// TwinCAT 3 PLC project TEXXX_XXX
// ProgramVersion: 3.1.4024.0
// libraries:
//   Tc2_Standard, * (Beckhoff Automation GmbH)
//   Tc2_System, * (Beckhoff Automation GmbH)
//   Tc2_Utilities, * (Beckhoff Automation GmbH)
//   Tc3_Module, * (Beckhoff Automation GmbH)
// project tree:
//   DUTs/HMI/ ST_StatusBanner.TcDUT (not stored), ST_Timers.TcDUT (not stored)
//   DUTs/IO/CARDS/ ST_Terminal_Info.TcDUT (not stored), ST_EL1809.TcDUT (not stored), ST_EL2809.TcDUT (not stored)
//   DUTs/MASTER/ E_MachineState.TcDUT (not stored), E_ProcessCycle.TcDUT (not stored), ST_ButtonsLamps.TcDUT (not stored), ST_HMI_IO.TcDUT (not stored), ST_MachineStatus.TcDUT (not stored), ST_MasterCTRL.TcDUT (not stored), ST_StationCMD.TcDUT (not stored), ST_StationStatus.TcDUT (not stored), ST_Puls.TcDUT (not stored), ST_StatisticsHMI.TcDUT (not stored)
//   DUTs/MASTER/log_CSV/ ST_CSVProcess.TcDUT, ST_UserLog.TcDUT (not stored), ST_CycleData.TcDUT (not stored)
//   DUTs/PDFMaker/ ST_EventsPDF.TcDUT, ST_EventsPdfConstants.TcDUT, ST_JavasCriptPDF.TcDUT, ST_PDFMaker.TcDUT
//   DUTs/STATIONS/STATION_1/ E_Station1_State.TcDUT (not stored), ST_CycleDataStation1.TcDUT (not stored), ST_Station_1.TcDUT (not stored)
//   DUTs/STATIONS/STATION_2/ E_Station2_State.TcDUT (not stored), ST_CycleDataStation2.TcDUT (not stored), ST_Station_2.TcDUT (not stored)
//   DUTs/STATIONS/STATION_3/ E_Station3_State.TcDUT (not stored), ST_CycleDataStation3.TcDUT (not stored), ST_Station_3.TcDUT (not stored)
//   DUTs/USER_ALARMS_EVENTS/EVENTS/ ST_ActiveEvents.TcDUT (not stored), ST_EventsAssigment.TcDUT (not stored), ST_EventsAssigmentGeneral.TcDUT (not stored), ST_EventsHistory.TcDUT, ST_EVENT.TcDUT (not stored), ST_StationEvents.TcDUT (not stored)
//   DUTs/USER_ALARMS_EVENTS/ ST_UserLogHMI.TcDUT (not stored)
//   GVLs/ GVL_Constants.TcGVL, GVL_HMI.TcGVL, GVL_IO.TcGVL (not stored), GVL_Master.TcGVL, GVL_Persistent.TcGVL, GVL_Stations.TcGVL (not stored)
//   / PlcTask.TcTTO (not stored)
//   POUs/A_MASTER/ A_1_PRG_Main_Master.TcPOU, A_2_PRG_MachineCtrl.TcPOU (not stored), A_3_PRG_FaultHandling.TcPOU (not stored), A_4_PRG_MasterSystemTime.TcPOU (not stored)
//   POUs/B_STATIONS/B_1_LEAK_TEST/ B_1_1_PRG_Master_Station_1.TcPOU (not stored)
//   POUs/B_STATIONS/B_2_HEIGHT_TEST/ B_2_1_PRG_Master_Station_2.TcPOU
//   POUs/B_STATIONS/B_3_STATION_3/ B_3_1_PRG_Master_Station_3.TcPOU (not stored)
//   POUs/C_HMI/ C_1_PRG_MainHMI.TcPOU (not stored)
//   POUs/ MAIN.TcPOU (not stored)
//   POUs/Utilities/ FB_EventsManager.TcPOU, FB_PDFMaker.TcPOU, FB_UserLog.TcPOU (not stored), FB_Pulse.TcPOU (not stored), FB_TerminalInfo.TcPOU (not stored), FB_TimeControl.TcPOU (not stored), FB_WriteDataToCSV.TcPOU, PRG_Puls.TcPOU (not stored)
// real-time tasks:
//   TASK PlcTask: cycle T#10ms, priority 20, ADS port 350

// ---- DUTs/MASTER/log_CSV/ST_CSVProcess.TcDUT
TYPE ST_CSVProcess :
STRUCT
	
	//INPUTS
	bWriteData			: BOOL;
	bWriteCSV			: BOOL;
	sFileNamePath		: STRING(255);
	sDate				: STRING(255);
	aDataHistoryArrayLength : DINT;
	nMAX_CSV_ROWS		: UDINT;
	nMAX_CSV_COLUMNS	: UDINT;

	//OUTPUTS
	bError				: BOOL;
	bBusy				: BOOL;
	
	
	
	
END_STRUCT
END_TYPE

// ---- DUTs/PDFMaker/ST_EventsPDF.TcDUT
TYPE ST_EventsPDF :
STRUCT
	
	     sEvents				: STRING;
         sType					: STRING;
         sDate					: STRING;
         sTime					: STRING;

	
END_STRUCT
END_TYPE

// ---- DUTs/PDFMaker/ST_EventsPdfConstants.TcDUT
TYPE ST_EventsPdfConstants :
STRUCT
	
	sMachineName			: STRING(255);
	sUser					: STRING(255);
	sGroup					: STRING(255);
	sFileName				: STRING(255);
	
END_STRUCT
END_TYPE

// ---- DUTs/PDFMaker/ST_JavasCriptPDF.TcDUT
TYPE ST_JavasCriptPDF :
STRUCT
	
	stEventsPDF				: ARRAY [0..2000] OF ST_EventsPDF;
	stEventsPdfConstants	: ST_EventsPdfConstants;
	bMakePDF				: BOOL;
	
	
END_STRUCT
END_TYPE

// ---- DUTs/PDFMaker/ST_PDFMaker.TcDUT
TYPE ST_PDFMaker :
STRUCT
	
	//INPUTS
	bWriteData			: BOOL;
	sDate				: STRING(255);
	aDataHistoryArrayLength : DINT;
	nDataHistoryIndex	: DINT;
	

	//OUTPUTS
	
	sFileName			: STRING(255);
	bDataWrited			: BOOL;
	

END_STRUCT
END_TYPE

// ---- DUTs/USER_ALARMS_EVENTS/EVENTS/ST_EventsHistory.TcDUT
TYPE ST_EventsHistory :
STRUCT
	
	sEventTex									: STRING(255);
	sType										: STRING(255);
	sDate										: STRING(255);
	sTime										: STRING(255);
	nEventsAmount								: DINT;
	abType										: DINT;					//1:Alarm
																		//2:Alert
																		//3:Message
	
END_STRUCT
END_TYPE

// ---- GVLs/GVL_Constants.TcGVL
VAR_GLOBAL CONSTANT
////////////////////////////////////////:	///////////////////////////////////////////////////
/////////////////////////////////////////////////////////////////////////////////////HMI/////////////////////////////////////////////////////////////////////////////////////
	
    sWHITE                              :   STRING(40)  := '{"color":"rgba(255,255,255,255)"}';
    sBLACK                              :   STRING(40)  := '{"color":"rgba(0,0,0,1)"}';
    sYELLOW                             :   STRING(40)  := '{"color":"rgba(255,255,0,1)"}';
    sGREEN                             	:   STRING(40)  := '{"color":"rgba(70,166,63,1)"}';
	sLGREEN                             :   STRING(40)  := '{"color":"rgba(58,211,20,1)"}';
    sORANGE                             :   STRING(40)  := '{"color":"rgba(255,153,51,1)"}';
    sNYPROORANGE                        :   STRING(40)  := '{"color":"rgba(255,140,0,1)"}';
    sRED                                :   STRING(40)  := '{"color":"rgba(255,0,0,1)"}';
	sLRED                               :   STRING(40)  := '{"color":"rgba(233,53,44,1)"}';
    sBLUE                               :   STRING(40)  := '{"color":"rgba(0,0,255,1)"}';
	sLBLUE                              :   STRING(40)  := '{"color":"rgba(0,162,232,1)"}';
    sGREY                               :   STRING(40)  := '{"color":"rgba(164,158,158,1)"}';
    sScreenGREY                         :   STRING(40)  := '{"color":"rgba(225,225,225,1)"}';
    sDARKGREY                           :   STRING(40)  := '{"color":"rgba(50,50,50,1)"}';
    sPURPLE                             :   STRING(40)  := '{"color":"rgba(128,0,128,1)"}';
    sVIOLET                             :   STRING(40)  := '{"color":"rgba(204,153,255,1)"}';
    sTRANSP                             :   STRING(40)  := '{"color":"rgba(255,255,255,0)"}';
    sGREENPass                          :   STRING(40)  := '{"color":"rgba(0,153,51,1)"}';
    sREDFail                            :   STRING(40)  := '{"color":"rgba(244,68,68,255)"}';
    sBLUEInProgress                     :   STRING(40)  := '{"color":"rgba(54,100,221,1)"}';
	sGREENISHTEAColor					:	STRING(40)  := '{"color":"rgba(60,192,134,255)"}'	;		

	nBLACK								: 	DWORD 	:= 	16#FF000000;	 // format: TTRRGGBB where T -> 00 = full transparency and FF = full opaque
	nWHITE								: 	DWORD 	:= 	16#FFFFFFFF;
	nYELLOW								: 	DWORD 	:= 	16#FFFFFF00; 
	nGREEN								: 	DWORD 	:= 	16#FF008A00;
	nLIGHTGREEN                         :   DWORD   :=  16#FF98FB89;
	nORANGE								: 	DWORD 	:= 	16#FFFFA500;
	nNYPROORANGE						:	DWORD	:=	16#FFF05322;
	nRED								: 	DWORD 	:= 	16#FFFF0000;
	nBLUE								: 	DWORD 	:= 	16#FF0000FF;
	nLIGHTBLUE                          :   DWORD   :=  16#FF08ADF4;
	nGREY								: 	DWORD 	:= 	16#FFA9A9A9;	
	nDARKGREY							:	DWORD	:=	16#FF808080;
	nPURPLE								:	DWORD	:=	16#FF800080;
	nVIOLET								:	DWORD	:=	16#FFEE82EE;
	nTRANSP								:	DWORD	:=	16#00FFFFFF;	// full transparent WHITE
	
/////////////////////////////////////////////////////////////////////////////////////CSV/////////////////////////////////////////////////////////////////////////////////////
	

	
	
	
END_VAR

// ---- GVLs/GVL_HMI.TcGVL
VAR_GLOBAL
////////////////////////////////////////:	///////////////////////////////////////////////////
/////////////////////////////////////////////////////////////////////////////////////GENERIC/////////////////////////////////////////////////////////////////////////////////////

	stHMI_IO							: ST_HMI_IO;
	bQuitHMI							: BOOL;
	bShutDown							: BOOL;
	stStatusBanner						: ST_StatusBanner;
	rOpenPopUp							: R_TRIG;
	nPopUp								: DINT;
	
	

/////////////////////////////////////////////////////////////////////////////////////SYSTEM INFO/////////////////////////////////////////////////////////////////////////////////////

	sSoftwareVersion					: STRING := ' 1.0 ';
	sSoftwareDate						: STRING := ' 10.December.2024 ';
	sTC3Version							: STRING := ' v3.1.4024.53, Runtime v3.1.4024.40 ';
	sHMIVersion							: STRING := ' TcXaeShell Version 15.0.28010.2050 D15.8 ';
	sSystemName							: STRING := ' Print & Applay Labeller ' ;
	sProjectID							: STRING := ' TE 1099 PAL' ;
	sAplication                     	: STRING := ' Print & Applay Labeller ';
	sHMIServer                			: STRING := ' ---- ';
	
	NetAmsId        	       			: T_AmsNetId := ''; // AMS-ID for com port setup 
	
/////////////////////////////////////////////////////////////////////////////////////USER LOG/////////////////////////////////////////////////////////////////////////////////////

	sUserGroupIn						: STRING;
	sUserGroupOut						: STRING;
	sUserName							: STRING;
	bUserLoggedIn						: BOOL;			
	bLogOut								: BOOL;	
	rUserLoggedIn						: R_TRIG;

/////////////////////////////////////////////////////////////////////////////////////MANUAL/////////////////////////////////////////////////////////////////////////////////////

	bEnableManual						: BOOL;
	nMainRegion							: DINT;
	bManualModeOffFlag					: BOOL;
	
END_VAR

// ---- GVLs/GVL_Master.TcGVL
VAR_GLOBAL
////////////////////////////////////////:	///////////////////////////////////////////////////
/////////////////////////////////////////////////////////////////////////////////////GENERIC/////////////////////////////////////////////////////////////////////////////////////

	// PowerUP 
	tonSystemPowerUP				:TON;
	tSystemPowerUP_Time				:TIME								:=T#35S;
	bSystemPoweringUP				:BOOL								:=TRUE; //Global System PowerUP Flag
	
	fbSystemShutDown     	        : NT_Shutdown;
	stButtonsLamps					: ST_ButtonsLamps;
	stPuls							: ST_Puls;		

	stCSVProcess					: ST_CSVProcess;
/////////////////////////////////////////////////////////////////////////////////////Event Log/////////////////////////////////////////////////////////////////////////////////////
	
	stStationEvents				: ARRAY[0..3] OF  ST_StationEvents;//0: GENERAL
																	//1: STATION 1
																	//1: STATION 2
																	//3: STATION 3
	astActiveEvents				: ARRAY [0..50] OF ST_ActiveEvents;
	stEventsAssigment			: ST_EventsAssigmentGeneral;

/////////////////////////////////////////////////////////////////////////////////////MACHINE CONTROL////////////////////////////////////////////////////////////////////////////
	
	stMachineStatus					: ST_MachineStatus;	
	stMasterCtrl					: ST_MasterCTRL;
	bStatisticsTest					: ARRAY[0..6] OF  BOOL;
	
////////////////////////////////////////////////////////////////////////////////////SYSTEM////////////////////////////////////////////////////////////////////////////
	stSystemTime				: TIMESTRUCT;
	sSystemTime					: STRING(255);
	sSystemDate					: STRING(255);
	
	bResetTest								: BOOL;
	tonResetTest							: TON;
	
END_VAR

// ---- GVLs/GVL_Persistent.TcGVL

VAR_GLOBAL PERSISTENT
	
/////////////////////////////////////////////////////////////////////////////////////Log/////////////////////////////////////////////////////////////////////////////////////
	
	stUserLog					: ARRAY [0..250] OF ST_UserLog;
	
	stStatisticsHMI				: ARRAY [0..3] OF ST_StatisticsHMI;	//0: GENERAL
																	//1: STATION 1
																	//2: STATION 2
																	//3: STATION 3
	aDataHistory				: ARRAY[0..200] OF ST_CycleData;
	nIndexDataHistory			: DINT;
	astEventsHistory			: ARRAY[0..200] OF ST_EventsHistory;
	stJavasCriptPDF				: ST_JavasCriptPDF;


END_VAR

// ---- POUs/A_MASTER/A_1_PRG_Main_Master.TcPOU
PROGRAM A_1_PRG_Main_Master
VAR
	
	rtrigButton             				: ARRAY[1..3] OF Tc2_Standard.R_TRIG;
	ftrigButton             				: ARRAY[1..3] OF Tc2_Standard.F_TRIG; 
	
	fbStringFormatter       				: Tc2_Utilities.FB_FormatString;
	fbEventsManager							: FB_EventsManager;
	
	ntShutdown								: TC2_Utilities.NT_Shutdown;
	closeChrome 							: NT_StartProcess;
	tonUserLogOut							: TON;
	fbUserLog								: FB_UserLog;
	
	nFindAdm								: INT;
	nFindEng								: INT;
	nFindOpe								: INT;
	sUserGroupName							: STRING (255);
	sAdmGroup								: STRING (255)							:= 'Administrator';
	sEngGroup								: STRING (255)							:= 'Engineer';
	sOpeGroup								: STRING (255)							:= 'Operator';
	
	rEfficency								: STRING(510);
	
	fbSystemTime							: NT_GetTime;
	
////////////////////////////////////////////////////////////////////////////////////CSV////////////////////////////////////////////////////////////////////////////	

	//stEventsCSVProcess						:  ST_CSVProcess;
	//fbWriteDataToCSV_Events					: FB_WriteDataToCSV;
	fbPDFMaker								: FB_PDFMaker;
	stPDFMaker								: ST_PDFMaker;
	i										: DINT;
	

	
END_VAR

/////////////////////////////////////////////////////////////////////////////////////GENERAL/////////////////////////////////////////////////////////////////////////////////////
A_3_PRG_FaultHandling();
a_ACT_ButtonsLamps();
b_ACT_PDFMaker();
d_ACT_ShutdownAndQuit();
e_ACT_UserLog();
f_ACT_TerminalInfo();
g_ACT_Manual();
h_ACT_Statistics();

C_1_PRG_MainHMI();
//D_1_1_PROG_Write_Data_To_CSV();
//D_2_1_PROG_Write_Data_To_CSV();

PRG_Puls();

// System PowerUP CTRL
tonSystemPowerUP(IN:=bSystemPoweringUP, PT:=tSystemPowerUP_Time);
IF tonSystemPowerUP.Q THEN 
bSystemPoweringUP:=FALSE;
END_IF


A_4_PRG_MasterSystemTime();
/////////////////////////////////////////////////////////////////////////////////////STATIONS/////////////////////////////////////////////////////////////////////////////////////

B_1_1_PRG_Master_Station_1(CMD := CMD_Station1);
B_2_1_PRG_Master_Station_2(CMD := CMD_Station2);
B_3_1_PRG_Master_Station_3(CMD := CMD_Station3);

/////////////////////////////////////////////////////////////////////////////////////PROCESS/////////////////////////////////////////////////////////////////////////////////////

A_2_PRG_MachineCtrl();

/////////////////////////////////////////////////////////////////////////////////////EVENT LOG/////////////////////////////////////////////////////////////////////////////////////

fbEventsManager	(			//INPUTS
							bPulse 							:= stPuls.bFlash10Hz, 
							bResetFaults 					:= bResetTest, 
							stStationEvents 				:= stStationEvents,
							sSystemTime						:= sSystemTime,
							sSystemDate						:= sSystemDate,
 							stEventsAssigment				:= stEventsAssigment,
							bDataWritedInCSV				:= stPDFMaker.bDataWrited,
							
							//OUTPUTS
							astActiveEvents 				=> astActiveEvents,
							astEventsHistory				=> astEventsHistory,
							bWriteDataInCSV					=> stPDFMaker.bWriteData,
							nDataHistoryIndex				=> stPDFMaker.nDataHistoryIndex
							);



////////////////////////////////////////////////////////////////////////////////////SYSTEM DATE & TIME/////////////////////////////////////////////////////////////////////////////////////

fbSystemTime( START := stPuls.bFlash10Hz, TIMESTR => stSystemTime);
	

sSystemTime					:= 	CONCAT( STR1 := WORD_TO_STRING(stSystemTime.wHour), STR2 := CONCAT( STR1 := ':', STR2 := 
								CONCAT( STR1 := WORD_TO_STRING(stSystemTime.wMinute), STR2 := 
								CONCAT(STR1 := ':', STR2 := WORD_TO_STRING(stSystemTime.wSecond)))));
								
sSystemDate					:= 	CONCAT( STR1 := WORD_TO_STRING(stSystemTime.wDay), STR2 := 
								CONCAT(STR1 := '/', STR2 := CONCAT(STR1 := WORD_TO_STRING(stSystemTime.wMonth), STR2 := 
								CONCAT(STR1 := '/', STR2 := WORD_TO_STRING(stSystemTime.wYear)))));

ACTION a_ACT_ButtonsLamps:
//===================================================================
stButtonsLamps.bStartButtonFallingEdge 	:= ftrigButton[1].Q ;
stButtonsLamps.bStartButtonRisingEdge 	:= rtrigButton[1].Q ;
stButtonsLamps.bStopButtonFallingEdge 	:= ftrigButton[2].Q ; 
stButtonsLamps.bStopButtonRisingEdge 	:= rtrigButton[2].Q ;  
stButtonsLamps.bResetButtonFallingEdge 	:= ftrigButton[3].Q ;
stButtonsLamps.bResetButtonRisingEdge 	:= rtrigButton[3].Q ;



ftrigButton[1](CLK :=);
rtrigButton[1](CLK						:=);
ftrigButton[2](CLK						:=);
rtrigButton[2](CLK						:=);
ftrigButton[3](CLK	:=bResetTest 		);
rtrigButton[3](CLK						:=);



//GVL_IO.dw_T11_EL2809.qRESETButton_Indicator := stPuls.bFlash2Hz AND (NOT stMachineStatus.bInitialising AND NOT stMachineStatus.bAutoCycle AND NOT stMachineStatus.bManualMode AND NOT stMachineStatus.bReadyToStart) ;
//GVL_IO.dw_T11_EL2809.qStartButton_Indicator := (stPuls.bFlash2Hz AND stMachineStatus.bReadyToStart) OR (stMachineStatus.bManualMode AND stPuls.bFlash4Hz ) ;
END_ACTION

ACTION b_ACT_PDFMaker:
//EVENTS TO CSV

fbPDFMaker(					
							aDataHistory				:= astEventsHistory,
							bWriteData					:= stPDFMaker.bWriteData,
							sDate						:= stPDFMaker.sDate,
							aDataHistoryArrayLength		:= 1000,
							nDataHistoryIndex			:= stPDFMaker.nDataHistoryIndex,
							sUser						:= 'sebastian',//sUserName,
							sGroup						:= 'administrator',//sUserGroupOut,
							sMachineName				:= 'example',
							
							bDataWrited					=> stPDFMaker.bDataWrited,
							stJavasCriptPDF				=> stJavasCriptPDF,
							bMakePdf					=> stJavasCriptPDF.bMakePDF
							);

(*stPDFMaker.sDate			:= 	CONCAT( STR1 := WORD_TO_STRING(stSystemTime.wDay), STR2 := 
								CONCAT(STR1 := '_', STR2 := CONCAT(STR1 := WORD_TO_STRING(stSystemTime.wMonth), STR2 := 
								CONCAT(STR1 := '_', STR2 := WORD_TO_STRING(stSystemTime.wYear)))));	*)
//CSV
(*fbWriteDataToCSV_Events( 	bWriteData					:= stEventsCSVProcess.bWriteData,
							sFileNamePath				:= stEventsCSVProcess.sFileNamePath,
							sDate						:= stEventsCSVProcess.sDate,
							aDataHistoryArrayLength		:= stEventsCSVProcess.aDataHistoryArrayLength,
							nMAX_CSV_ROWS				:= stEventsCSVProcess.nMAX_CSV_ROWS,
							nMAX_CSV_COLUMNS			:= stEventsCSVProcess.nMAX_CSV_COLUMNS,
							nDataHistoryIndex			:= stEventsCSVProcess.nDataHistoryIndex,
							
							bBusy						=> stEventsCSVProcess.bBusy,
							bError						=> stEventsCSVProcess.bError,
							nErrId						=>,
							bDataWrited					=> stEventsCSVProcess.bDataWrited,
							aDataHistory				:= astEventsHistory);
							

(*stEventsCSVProcess.sDate	:= 	CONCAT( STR1 := WORD_TO_STRING(stSystemTime.wDay), STR2 := 
								CONCAT(STR1 := '_', STR2 := CONCAT(STR1 := WORD_TO_STRING(stSystemTime.wMonth), STR2 := 
								CONCAT(STR1 := '_', STR2 := WORD_TO_STRING(stSystemTime.wYear)))));		*)				
								

stEventsCSVProcess.sFileNamePath						:= 'C:\Users\Sebastian.Ulloa\Desktop\GIT PROJECTS\TEMPLATES\TEMPLATE_VER1\CSV\EVENTS\';								
stEventsCSVProcess.aDataHistoryArrayLength				:= 200;
stEventsCSVProcess.nMAX_CSV_ROWS						:= 1000;
stEventsCSVProcess.nMAX_CSV_COLUMNS						:= 4;*)
END_ACTION

ACTION d_ACT_ShutdownAndQuit:
closeChrome(
    NetId := '',
    PathStr := 'C:\Windows\System32\mshta vbscript:Execute("CreateObject(""WScript.Shell"").Run ""powershell -c',
    DirName := 'C:\Windows\System32\WindowsPowerShell\v1.0',
    ComndLine := 'taskkill /F /IM chrome.exe /T"", 0: window.close")',
    Start := bQuitHmi,
    TmOut := DEFAULT_ADS_TIMEOUT
);
 
bQuitHmi:= FALSE;

ntShutdown(NETID := NetAmsId, DELAY := 5, START := bShutDown);
END_ACTION

ACTION e_ACT_UserLog:
sUserGroupName																:= sUserGroupIn;

nFindAdm	:= TC2_Utilities.FIND( 	STR1									:= sUserGroupName,
									STR2									:= sAdmGroup);
									
nFindEng	:= TC2_Utilities.FIND( 	STR1									:= sUserGroupName,
									STR2									:= sEngGroup);
					
nFindOpe	:= TC2_Utilities.FIND( 	STR1									:= sUserGroupName,
									STR2									:= sOpeGroup);
				
IF nFindAdm <> 0 THEN
	sUserGroupOut															:= 'Administrator';
ELSIF nFindEng <> 0 THEN
	sUserGroupOut															:= 'Engineer';
ELSIF nFindOpe <> 0 THEN
	sUserGroupOut															:= 'Operator';
ELSE sUserGroupOut															:= '';
END_IF

tonUserLogOut( IN := (sUserGroupOut <> 'Administrator' OR sUserGroupOut <> 'Engineer') AND bUserLoggedIn , PT := T#10M);

IF tonUserLogOut.Q THEN
	bLogOut 											:= TRUE;
ELSE bLogOut 											:= FALSE;
END_IF

rUserLoggedIn( CLK := bUserLoggedIn);

fbUserLog(	nNumberOfData								:= 250,
			bSaveSignal									:= rUserLoggedIn.Q, 
			sUser										:= sUserName,
			sGroup										:= sUserGroupOut,
			sDate										:= sSystemDate,
			sTime										:= sSystemTime,
			aDataOutput									:= stUserLog);
END_ACTION

ACTION f_ACT_TerminalInfo:
dw_T03_EL1809.stTerminalInfo.fbTerminalInfo( 	nTerminalState						:= dw_T03_EL1809.stTerminalInfo.nTerminal_State,
												sTerminalState						=> dw_T03_EL1809.stTerminalInfo.sTerminalInfo);
												
dw_T04_EL2809.stTerminalInfo.fbTerminalInfo(	nTerminalState						:= dw_T04_EL2809.stTerminalInfo.nTerminal_State,
												sTerminalState						=> dw_T04_EL2809.stTerminalInfo.sTerminalInfo);
END_ACTION

ACTION g_ACT_Manual:


IF stMachineStatus.bReadyToStart THEN
	bEnableManual											:= TRUE;
ELSE bEnableManual											:= FALSE;
END_IF

IF nMainRegion = 5 AND stMasterCtrl.bNoImmediateFault AND stMasterCtrl.bNoCycleStopFault
	AND NOT stMasterCtrl.bCycleStopRequest AND NOT stButtonsLamps.bStopButtonFallingEdge THEN
	stMasterCtrl.bManualModeRequest							:= TRUE;
	bManualModeOffFlag										:= FALSE;
ELSE 
	stMasterCtrl.bManualModeRequest							:= FALSE; 
	bManualModeOffFlag										:= TRUE;											
END_IF
END_ACTION

ACTION h_ACT_Statistics:
stStatisticsHMI[0].sName			:= 'TOTAL';

stStatisticsHMI[0].nGood		:= stStatisticsHMI[1].nGood + stStatisticsHMI[2].nGood + stStatisticsHMI[3].nGood;
stStatisticsHMI[0].nTotalGood	:= stStatisticsHMI[1].nTotalGood + stStatisticsHMI[2].nTotalGood + stStatisticsHMI[3].nTotalGood;
stStatisticsHMI[0].nBad			:= stStatisticsHMI[1].nBad + stStatisticsHMI[2].nBad + stStatisticsHMI[3].nBad;
stStatisticsHMI[0].nTotalBad	:= stStatisticsHMI[1].nTotalBad + stStatisticsHMI[2].nTotalBad + stStatisticsHMI[3].nTotalBad;

								

IF (( stStatisticsHMI[0].nGood + stStatisticsHMI[0].nBad) <> 0) THEN
	
	rEfficency							:= LREAL_TO_FMTSTR(in := (DINT_TO_REAL(stStatisticsHMI[0].nGood) /( DINT_TO_REAL(stStatisticsHMI[0].nGood) + DINT_TO_REAL(stStatisticsHMI[0].nBad))) * 100.0,iPrecision := 2, bRound := TRUE);
	stStatisticsHMI[0].nEfficency		:= CONCAT(STR1 := '%', STR2 := (rEfficency));

ELSE stStatisticsHMI[0].nEfficency		:= CONCAT(STR1 := '%', STR2 := (DINT_TO_STRING(0)));
	
END_IF
END_ACTION

END_PROGRAM

// ---- POUs/Utilities/FB_EventsManager.TcPOU
FUNCTION_BLOCK FB_EventsManager

VAR_INPUT
	
	bPulse					: BOOL;
	sSystemTime				: STRING(255);
	sSystemDate				: STRING(255);
	bDataWritedInCSV		: BOOL;
	
END_VAR

VAR_OUTPUT

	astActiveEvents			: ARRAY [0..50] OF ST_ActiveEvents;
	astEventsHistory		: ARRAY[0..200] OF ST_EventsHistory;
	bWriteDataInCSV			: BOOL;
	nDataHistoryIndex		: DINT;
	

END_VAR

VAR
	
	i								: ARRAY [0..1] OF DINT;
	j								: ARRAY [0..1] OF DINT;
	m								: ARRAY [0..3] OF DINT;
	k								: ARRAY [0..1] OF DINT;
	l								: DINT;
	n								: DINT;
	
	bEventsAssigmentSignal			: BOOL		:= TRUE;
	
	

	
END_VAR

VAR_IN_OUT
	
	stStationEvents			: ARRAY[0..3] OF ST_StationEvents;
	stEventsAssigment		: ST_EventsAssigmentGeneral;
	bResetFaults			: BOOL;
	
END_VAR

ACT_FaultTrig();
ACT_ActiveEvents_DataHistory();


IF bEventsAssigmentSignal THEN
	ACT_EventTextAssigment();
	bEventsAssigmentSignal := FALSE;
END_IF

ACTION ACT_ActiveEvents_DataHistory:
IF bPulse AND NOT bWriteDataInCSV THEN

FOR k[0] := 0 TO 3 DO
	
	FOR k[1] := 0 TO 100 DO
		
		IF stStationEvents[k[0]].aEvents[k[1]].bImmediateFault AND stStationEvents[k[0]].aEvents[k[1]].bEventFlag AND NOT stStationEvents[k[0]].aEvents[k[1]].bActive THEN
			
			//ACTIVE EVENTS
			astActiveEvents[l].sEventTex				:= 	stStationEvents[k[0]].aEvents[k[1]].bEventTextHMI;
			astActiveEvents[l].sType					:= 'Immediate Fault';						
			astActiveEvents[l].abType					:= 1; 
			astActiveEvents[l].sSolution				:= stStationEvents[k[0]].aEvents[k[1]].sSolution;
			stStationEvents[k[0]].aEvents[k[1]].bActive := TRUE;
			
			//EVENTS HISTORY
			FOR n := 199 TO 0 BY -1 DO
							
				astEventsHistory[n+1].sEventTex				:= astEventsHistory[n].sEventTex;
				astEventsHistory[n+1].sType					:= astEventsHistory[n].sType;
				astEventsHistory[n+1].abType				:= astEventsHistory[n].abType;
				astEventsHistory[n+1].sDate					:= astEventsHistory[n].sDate;										
				astEventsHistory[n+1].sTime					:= astEventsHistory[n].sTime;
				
			END_FOR

			astEventsHistory[0].sEventTex				:= stStationEvents[k[0]].aEvents[k[1]].bEventTextHMI;
			astEventsHistory[0].sType					:= 'Immediate Fault';
			astEventsHistory[0].abType					:= 1;
			astEventsHistory[0].sDate					:= 	sSystemDate;										
			astEventsHistory[0].sTime					:= 	sSystemTime;
			l											:= l + 1;			
			nDataHistoryIndex							:= 1 + nDataHistoryIndex;		
			
		END_IF
		
		IF stStationEvents[k[0]].aEvents[k[1]].bCycleStopFault AND stStationEvents[k[0]].aEvents[k[1]].bEventFlag AND NOT stStationEvents[k[0]].aEvents[k[1]].bActive THEN
			
			//ACTIVE EVENTS
			astActiveEvents[l].sEventTex				:= 	stStationEvents[k[0]].aEvents[k[1]].bEventTextHMI;
			astActiveEvents[l].sType					:= 'Cycle Stop Fault';						
			astActiveEvents[l].abType					:= 1; 
			astActiveEvents[l].sSolution				:= stStationEvents[k[0]].aEvents[k[1]].sSolution;
			stStationEvents[k[0]].aEvents[k[1]].bActive := TRUE;
			
			//EVENTS HISTORY
			FOR n := 199 TO 0 BY -1 DO
							
				astEventsHistory[n+1].sEventTex				:= astEventsHistory[n].sEventTex;
				astEventsHistory[n+1].sType					:= astEventsHistory[n].sType;
				astEventsHistory[n+1].abType				:= astEventsHistory[n].abType;
				astEventsHistory[n+1].sDate					:= astEventsHistory[n].sDate;										
				astEventsHistory[n+1].sTime					:= astEventsHistory[n].sTime;
				
			END_FOR
			
			astEventsHistory[0].sEventTex				:= stStationEvents[k[0]].aEvents[k[1]].bEventTextHMI;
			astEventsHistory[0].sType					:= 'Cycle Stop Fault';
			astEventsHistory[0].abType					:= 1;
			astEventsHistory[0].sDate					:= 	sSystemDate;										
			astEventsHistory[0].sTime					:= 	sSystemTime;
															
			l											:= l + 1;		
			nDataHistoryIndex							:= 1 + nDataHistoryIndex;	
					
		END_IF
		
		IF stStationEvents[k[0]].aEvents[k[1]].bCycleStopRequest AND stStationEvents[k[0]].aEvents[k[1]].bEventFlag AND NOT stStationEvents[k[0]].aEvents[k[1]].bActive THEN
			
			//ACTIVE EVENTS
			astActiveEvents[l].sEventTex				:= 	stStationEvents[k[0]].aEvents[k[1]].bEventTextHMI;
			astActiveEvents[l].sType					:= 'Cycle Stop Request';						
			astActiveEvents[l].abType					:= 2; 
			astActiveEvents[l].sSolution				:= stStationEvents[k[0]].aEvents[k[1]].sSolution;
			stStationEvents[k[0]].aEvents[k[1]].bActive := TRUE;
			
			//EVENTS HISTORY
			FOR n := 199 TO 0 BY -1 DO
							
				astEventsHistory[n+1].sEventTex				:= astEventsHistory[n].sEventTex;
				astEventsHistory[n+1].sType					:= astEventsHistory[n].sType;
				astEventsHistory[n+1].abType				:= astEventsHistory[n].abType;
				astEventsHistory[n+1].sDate					:= astEventsHistory[n].sDate;										
				astEventsHistory[n+1].sTime					:= astEventsHistory[n].sTime;
				
			END_FOR

			astEventsHistory[0].sEventTex				:= stStationEvents[k[0]].aEvents[k[1]].bEventTextHMI;
			astEventsHistory[0].sType					:= 'Cycle Stop Request';
			astEventsHistory[0].abType					:= 2;
			astEventsHistory[0].sDate					:= 	sSystemDate;										
			astEventsHistory[0].sTime					:= 	sSystemTime;
															
			l											:= l + 1;	
			nDataHistoryIndex							:= 1 + nDataHistoryIndex;	
						
		END_IF
		
		IF stStationEvents[k[0]].aEvents[k[1]].bMessage AND stStationEvents[k[0]].aEvents[k[1]].bEventFlag AND NOT stStationEvents[k[0]].aEvents[k[1]].bActive THEN
			
			//ACTIVE EVENTS
			astActiveEvents[l].sEventTex				:= 	stStationEvents[k[0]].aEvents[k[1]].bEventTextHMI;
			astActiveEvents[l].sType					:= 'Message';						
			astActiveEvents[l].abType					:= 3; 
			astActiveEvents[l].sSolution				:= stStationEvents[k[0]].aEvents[k[1]].sSolution;
			stStationEvents[k[0]].aEvents[k[1]].bActive := TRUE;
			
			//EVENTS HISTORY
			FOR n := 199 TO 0 BY -1 DO
							
				astEventsHistory[n+1].sEventTex				:= astEventsHistory[n].sEventTex;
				astEventsHistory[n+1].sType					:= astEventsHistory[n].sType;
				astEventsHistory[n+1].abType				:= astEventsHistory[n].abType;
				astEventsHistory[n+1].sDate					:= astEventsHistory[n].sDate;										
				astEventsHistory[n+1].sTime					:= astEventsHistory[n].sTime;
				
			END_FOR

			astEventsHistory[0].sEventTex				:= stStationEvents[k[0]].aEvents[k[1]].bEventTextHMI;
			astEventsHistory[0].sType					:= 'Message';
			astEventsHistory[0].abType					:= 3;
			astEventsHistory[0].sDate					:= 	sSystemDate;										
			astEventsHistory[0].sTime					:= 	sSystemTime;
															
			l											:= l + 1;
			nDataHistoryIndex							:= 1 + nDataHistoryIndex;
										
		END_IF
		
		
	END_FOR

END_FOR

ELSIF bResetFaults THEN
	FOR l := 0 TO 50 DO
	
			astActiveEvents[l].sEventTex			:= 	'';
			astActiveEvents[l].sType				:= '';						
			astActiveEvents[l].abType				:= 0; 
			astActiveEvents[l].sSolution			:= '';
			
	END_FOR	
	
	FOR k[0] := 0 TO 3 DO
	
		FOR k[1] := 0 TO 100 DO
	
			stStationEvents[k[0]].aEvents[k[1]].bActive	:= FALSE;
		END_FOR
	END_FOR
	
	l												:= 0;
	k[0]											:= 0;
	k[1]											:= 0;	
	bResetFaults									:= FALSE;
ELSE
	
	k[0]											:= 0;
	k[1]											:= 0;
	
END_IF

IF nDataHistoryIndex = 201 THEN
	
	bWriteDataInCSV									:= TRUE;

END_IF 
	
IF bDataWritedInCSV THEN
	
	bWriteDataInCSV									:= FALSE;
	nDataHistoryIndex								:= 0;
	
END_IF


//



																		//0:Immediate Fault
																		//1:Cycle Stop Fault
																		//2: Cycle Stop Request
																		//3: Message
END_ACTION

ACTION ACT_EventTextAssigment:

FOR j[0] := 0 TO 3 DO
	
	FOR j[1] := 0 TO 100 DO 
		
		IF stStationEvents[j[0]].aEvents[j[1]].bImmediateFault THEN
			
			m[0]											:= m[0]+1;
			
			stStationEvents[j[0]].aEvents[j[1]].bEventTextHMI	:= 		CONCAT( STR1 := 'Immediate Fault N ', STR2 := 
																CONCAT( STR1 := DINT_TO_STRING(m[0]), str2 := 
																CONCAT( STR1 :=' - Station ' , STR2 := 
																CONCAT( STR1 := DINT_TO_STRING(j[0]), STR2 := 
																CONCAT( STR1 :=' - ', str2 := stStationEvents[j[0]].aEvents[j[1]].bEventText )))));
			stStationEvents[j[0]].aEvents[j[1]].bAssignedID	:= 	m[0];				
			
			//EVENTS ASSIGMENT
			stEventsAssigment.astImmediateFaultEvents[m[0]].sEventText	:= stStationEvents[j[0]].aEvents[j[1]].bEventTextHMI;
			stEventsAssigment.astImmediateFaultEvents[m[0]].sSolution	:= stStationEvents[j[0]].aEvents[j[1]].sSolution;
			
		ELSIF stStationEvents[j[0]].aEvents[j[1]].bCycleStopFault THEN
			
			m[1]											:= m[1]+1;
			
			stStationEvents[j[0]].aEvents[j[1]].bEventTextHMI	:= 		CONCAT( STR1 := 'Cycle Stop Fault N ', STR2 := 
																CONCAT( STR1 := DINT_TO_STRING(m[1]), str2 := 
																CONCAT( STR1 :=' - Station ' , STR2 := 
																CONCAT( STR1 := DINT_TO_STRING(j[0]), STR2 := 
																CONCAT( STR1 :=' - ', str2 := stStationEvents[j[0]].aEvents[j[1]].bEventText )))));
			stStationEvents[j[0]].aEvents[j[1]].bAssignedID	:= 	m[1];													
			
			//EVENTS ASSIGMENT
			stEventsAssigment.astCycleStopFaultEvents[m[1]].sEventText	:= stStationEvents[j[0]].aEvents[j[1]].bEventTextHMI;
			stEventsAssigment.astCycleStopFaultEvents[m[1]].sSolution	:= stStationEvents[j[0]].aEvents[j[1]].sSolution;
			
		ELSIF stStationEvents[j[0]].aEvents[j[1]].bCycleStopRequest THEN
		
			m[2]											:= m[2]+1;	
			
			stStationEvents[j[0]].aEvents[j[1]].bEventTextHMI	:= 		CONCAT( STR1 := 'Cycle Stop Request N ', STR2 := 
																CONCAT( STR1 := DINT_TO_STRING(m[2]), str2 := 
																CONCAT( STR1 :=' - Station ' , STR2 := 
																CONCAT( STR1 := DINT_TO_STRING(j[0]), STR2 := 
																CONCAT( STR1 :=' - ', str2 := stStationEvents[j[0]].aEvents[j[1]].bEventText )))));
			stStationEvents[j[0]].aEvents[j[1]].bAssignedID	:= 	m[2];													

			//EVENTS ASSIGMENT
			stEventsAssigment.astCycleStopRequestEvents[m[2]].sEventText	:= stStationEvents[j[0]].aEvents[j[1]].bEventTextHMI;
			stEventsAssigment.astCycleStopRequestEvents[m[2]].sSolution	:= stStationEvents[j[0]].aEvents[j[1]].sSolution;
			
		ELSIF stStationEvents[j[0]].aEvents[j[1]].bMessage THEN
			
			m[3]											:= m[3]+1;
			
			stStationEvents[j[0]].aEvents[j[1]].bEventTextHMI	:= 		CONCAT( STR1 := 'Message N ', STR2 := 
																CONCAT( STR1 := DINT_TO_STRING(m[3]), str2 := 
																CONCAT( STR1 :=' - Station ' , STR2 := 
																CONCAT( STR1 := DINT_TO_STRING(j[0]), STR2 := 
																CONCAT( STR1 :=' - ', str2 := stStationEvents[j[0]].aEvents[j[1]].bEventText )))));
			stStationEvents[j[0]].aEvents[j[1]].bAssignedID	:= 	m[3];													
				
			//EVENTS ASSIGMENT
			stEventsAssigment.astMessage[m[3]].sEventText	:= stStationEvents[j[0]].aEvents[j[1]].bEventTextHMI;
			stEventsAssigment.astMessage[m[3]].sSolution	:= stStationEvents[j[0]].aEvents[j[1]].sSolution;	
			
		END_IF
		
	END_FOR
	
	
END_FOR
j[0]														:= 0;
j[1]														:= 0;
m[0]														:= 0;
m[1]														:= 0;
m[2]														:= 0;
m[3]														:= 0;
END_ACTION

ACTION ACT_FaultTrig:
IF bPulse THEN
	

	FOR i[0] := 0 TO 3 DO
	//IMMEDIATE FAULT
		FOR i[1] :=0 TO 100 DO
			
			//IMMEDIATE FAULT
			IF stStationEvents[i[0]].aEvents[i[1]].bImmediateFault AND stStationEvents[i[0]].aEvents[i[1]].bEventFlag THEN
	
				stStationEvents[i[0]].bImmediateFault						:= TRUE;
		
			ELSIF bResetFaults THEN
				stStationEvents[i[0]].bImmediateFault						:= FALSE;
			END_IF
			//STOP FAULT
			IF stStationEvents[i[0]].aEvents[i[1]].bCycleStopFault AND stStationEvents[i[0]].aEvents[i[1]].bEventFlag THEN
	
				stStationEvents[i[0]].bCycleStopFault						:= TRUE;
		
			ELSIF bResetFaults THEN
				stStationEvents[i[0]].bCycleStopFault						:= FALSE;
			END_IF
		
			//STOP REQUEST
			IF stStationEvents[i[0]].aEvents[i[1]].bCycleStopRequest AND stStationEvents[i[0]].aEvents[i[1]].bEventFlag THEN
	
				stStationEvents[i[0]].bCycleStopRequest						:= TRUE;
		
			ELSIF bResetFaults THEN
				stStationEvents[i[0]].bCycleStopRequest						:= FALSE;
			END_IF
		
		END_FOR
	END_FOR

ELSE 	i[0]														:= 0;
		i[1]														:= 0;	
END_IF
END_ACTION

END_FUNCTION_BLOCK

// ---- POUs/Utilities/FB_PDFMaker.TcPOU
FUNCTION_BLOCK FB_PDFMaker
VAR_INPUT
	
	aDataHistory			: ARRAY[0..200] OF ST_EventsHistory;
	bWriteData				: BOOL;
	aDataHistoryArrayLength	: DINT;
	nDataHistoryIndex		: DINT;
	sDate					: STRING(255);
	
	sUser					: STRING(255);
	sGroup					: STRING(255);
	sMachineName			: STRING(255);
	
	 
END_VAR
VAR_OUTPUT
	
	stJavasCriptPDF		: ST_JavasCriptPDF;
	bDataWrited			: BOOL;
	bMakePdf			: BOOL;

END_VAR
VAR
	
	rWriteData				: R_TRIG;
	i						: DINT;
	nRowIndex				: DINT;
	sPDFDate				: STRING(255);
	sFileName				: STRING(255);
	tonResetData			: TON;
	
END_VAR

ACT_IO();
ACT_WriteData();

ACTION ACT_IO:
stJavasCriptPDF.stEventsPdfConstants.sGroup			:= sGroup;		
stJavasCriptPDF.stEventsPdfConstants.sMachineName	:= sMachineName;
stJavasCriptPDF.stEventsPdfConstants.sUser			:= sUser;
stJavasCriptPDF.stEventsPdfConstants.sFileName		:= sFileName;
END_ACTION

ACTION ACT_WriteData:
rWriteData( CLK := bWriteData);

IF rWriteData.Q THEN
	
	FOR i := 0 TO aDataHistoryArrayLength DO
				
					stJavasCriptPDF.stEventsPDF[nRowIndex + i].sEvents					:= 	aDataHistory[i].sEventTex;
					stJavasCriptPDF.stEventsPDF[nRowIndex + i].sType					:= 	aDataHistory[i].sType;
					stJavasCriptPDF.stEventsPDF[nRowIndex + i].sDate					:= 	aDataHistory[i].sDate;
					stJavasCriptPDF.stEventsPDF[nRowIndex + i].sTime					:= 	aDataHistory[i].sTime;
				
	END_FOR
	
	i													:= 0;
	
	bDataWrited											:= TRUE;
	nRowIndex											:= nRowIndex + 201;

	

END_IF

IF nDataHistoryIndex = 0 THEN
	
	bDataWrited											:= FALSE;

END_IF

IF sPDFDate <> sDate THEN
	
	bMakePdf							:= TRUE;
	sPDFDate							:= sDate;
	
END_IF

sFileName 								:= CONCAT( STR1 := 'PDF_', STR2 := sPDFDate);

tonResetData( IN := bMakePdf, PT := T#1S);

IF tonResetData.Q THEN
	
	FOR i := 0 TO 1000 DO
				
					stJavasCriptPDF.stEventsPDF[i].sDate					:= 	'';
					stJavasCriptPDF.stEventsPDF[i].sEvents					:=  '';
					stJavasCriptPDF.stEventsPDF[i].sTime					:= 	'';
					stJavasCriptPDF.stEventsPDF[i].sType					:= 	'';
				
	END_FOR
	nRowIndex 										:= 0;		
	bMakePdf										:= FALSE;
	i												:= 0;
END_IF
END_ACTION

END_FUNCTION_BLOCK

// ---- POUs/B_STATIONS/B_2_HEIGHT_TEST/B_2_1_PRG_Master_Station_2.TcPOU
PROGRAM B_2_1_PRG_Master_Station_2

VAR
	eState								: E_Station2_State;
	tonErrorReset						: TON;
	tonStationStopped					: TON;
	ctuErrorCounter						: CTU;
	rGoodStatistics						: R_TRIG;
	rBadStatistics						: R_TRIG;
	rEfficency							: STRING(510);
	
	bPersistentError					: BOOL;
	
	bEventsFlag							: ARRAY [0..100] OF BOOL;
/////////////////////////////////////////////////////////////////////////////////////I O/////////////////////////////////////////////////////////////////////////////////////	
	bStopped							: BOOL;
	bError								: BOOL;
	bReady								: BOOL;
	bDone								: BOOL;
	bPass								: BOOL;
	bFail								: BOOL;

	
END_VAR

VAR_INPUT	
	
	CMD									:ST_StationCMD;	
	
END_VAR

VAR_OUTPUT	
	
	STATUS								:ST_StationStatus;	
	
END_VAR

d_ACT_Set_Events_Station_2();
a_ACT_Ctrl_Station_2();
b_ACT_IO();
c_ACT_Statistics_Station_2();

ACTION a_ACT_Ctrl_Station_2:
/////////////////////////////////////////////////////////////////////////////////////UTILITIES/////////////////////////////////////////////////////////////////////////////////////
tonErrorReset( IN := (eState = E_Station2_State.RESET_ERROR), PT := T#500MS);
tonStationStopped( IN := bStopped, PT := T#1S);
ctuErrorCounter( CU := eState = E_Station2_State.RESET_ERROR, RESET := ((ctuErrorCounter.CV = 5) AND eState = E_Station2_State.PERSISTENT_ERROR), PV := 5, Q => bPersistentError);

/////////////////////////////////////////////////////////////////////////////////////CONDITIONS/////////////////////////////////////////////////////////////////////////////////////

IF (CMD.bAbort OR bError) AND ( eState			= E_Station2_State.HOMING OR
								eState			= E_Station2_State.READY OR
								eState			= E_Station2_State.MOVEMENT_A OR
								eState			= E_Station2_State.MOVEMENT_B OR
								eState			= E_Station2_State.MOVEMENT_C OR
								eState			= E_Station2_State.READY  OR
								eState			= E_Station2_State.DONE) THEN
								
	eState						:= E_Station2_State.STOPPING;
	
END_IF

CASE eState OF
	
	E_Station2_State.ABORTED:
								IF CMD.bEnable AND NOT bError THEN
									eState						:= E_Station2_State.HOMING;
								ELSIF bError THEN
									eState						:= E_Station2_State.ERROR;
								END_IF
	
	E_Station2_State.HOMING:
								IF bReady THEN
									eState						:= E_Station2_State.READY;
								END_IF
	E_Station1_State.RESET:
								stCycleDataStation2.bPass	:= FALSE;
								stCycleDataStation2.bFail	:= FALSE;
								
								eState						:= E_Station2_State.READY;
	E_Station2_State.READY:
								IF CMD.bExecute AND stStation2.Mov1 THEN
									eState						:= E_Station2_State.MOVEMENT_A;
								ELSIF CMD.bExecute AND stStation2.Mov2 THEN
									eState						:= E_Station2_State.MOVEMENT_B;
								ELSIF CMD.bExecute AND stStation2.Mov3 THEN
									eState						:= E_Station2_State.MOVEMENT_C;
								END_IF
	
	E_Station2_State.MOVEMENT_A:
								IF bDone AND stStation2.Mov1 THEN
									eState						:= E_Station2_State.DONE;
								END_IF
	
	E_Station2_State.MOVEMENT_B:
								IF bDone AND stStation2.Mov2 THEN
									eState						:= E_Station2_State.DONE;
								END_IF
	E_Station2_State.MOVEMENT_C:
								IF bDone AND stStation2.Mov3 THEN
									eState						:= E_Station2_State.DONE;
								END_IF
	E_Station2_State.DONE:
								IF  CMD.bReady THEN
									eState						:= E_Station2_State.READY;
								END_IF	
	E_Station1_State.RESULTS:
								
								IF bPass THEN
									stCycleDataStation2.bPass	:= TRUE;
								ELSIF bFail THEN
								 	stCycleDataStation2.bFail	:= TRUE;
								END_IF
								
								IF  CMD.bEndCycle THEN
									eState						:= E_Station2_State.RESET;
								END_IF
/////////////////////////////////////////////////////////////////////////////////////RESET CMD/////////////////////////////////////////////////////////////////////////////////////

	E_Station2_State.STOPPING: 
								IF tonStationStopped.Q THEN
									IF bError THEN
										eState						:= E_Station2_State.ERROR;
									ELSE eState						:= E_Station2_State.ABORTED;
									END_IF

								END_IF
	
	E_Station2_State.ERROR:
								IF NOT bError THEN
									eState						:= E_Station2_State.ABORTED;
								ELSE eState						:= E_Station2_State.RESET_ERROR;
								END_IF
	
	E_Station2_State.RESET_ERROR:
								IF tonErrorReset.Q AND NOT bPersistentError THEN
									eState						:= E_Station2_State.ERROR;
								ELSIF bPersistentError THEN
									eState						:= E_Station2_State.PERSISTENT_ERROR;
								END_IF
	
	E_Station2_State.PERSISTENT_ERROR:
								IF CMD.bReset THEN
									eState						:= E_Station2_State.ERROR;
								END_IF
								
								

ELSE eState := E_Station2_State.ABORTED;
	
END_CASE
/////////////////////////////////////////////////////////////////////////////////////STATUS/////////////////////////////////////////////////////////////////////////////////////

Status.bBusy				:= 	eState			= E_Station2_State.HOMING OR
								eState			= E_Station2_State.MOVEMENT_A OR
								eState			= E_Station2_State.MOVEMENT_B OR
								eState			= E_Station2_State.MOVEMENT_C OR
								eState			= E_Station2_State.STOPPING;
								
Status.bDone				:=	eState			= E_Station2_State.DONE;
											
Status.bError				:= 	eState			= (E_Station2_State.ERROR OR  E_Station2_State.RESET_ERROR OR E_Station2_State.PERSISTENT_ERROR);

Status.bReady				:= 	eState			= E_Station2_State.READY;

Status.bStopped				:= 	eState			= E_Station2_State.ABORTED OR
								eState			= E_Station2_State.READY OR
								eState			= E_Station2_State.ERROR OR
								eState			= E_Station2_State.RESET_ERROR;
END_ACTION

ACTION b_ACT_IO:
//bStopped								:=;
//bError								:=;
//bReady								:=;
//bDone
END_ACTION

ACTION c_ACT_Statistics_Station_2:
stStatisticsHMI[2].sName			:= 'Station 2';


rGoodStatistics( CLK := (stCycleDataStation2.bPass AND (eState = E_Station2_State.RESULTS)) OR bStatisticsTest[2]);
rBadStatistics( CLK := (stCycleDataStation2.bFail AND (eState = E_Station2_State.RESULTS)) OR bStatisticsTest[3]);

IF 	rGoodStatistics.Q THEN
	
	stStatisticsHMI[2].nGood		:= stStatisticsHMI[2].nGood + 1;
	stStatisticsHMI[2].nTotalGood	:= stStatisticsHMI[2].nTotalGood + 1;
	
END_IF
								
IF 	rBadStatistics.Q THEN
	
	stStatisticsHMI[2].nBad			:= stStatisticsHMI[2].nBad + 1;
	stStatisticsHMI[2].nTotalBad	:= stStatisticsHMI[2].nTotalBad + 1;
	
END_IF

IF stStatisticsHMI[2].bResetGood THEN
	stStatisticsHMI[2].nGood		:= 0;
END_IF

IF stStatisticsHMI[2].bResetBad THEN
	stStatisticsHMI[2].nBad			:= 0;
END_IF

IF (( stStatisticsHMI[2].nGood + stStatisticsHMI[2].nBad) <> 0) THEN
	
	rEfficency							:= LREAL_TO_FMTSTR(in := (DINT_TO_REAL(stStatisticsHMI[2].nGood) /( DINT_TO_REAL(stStatisticsHMI[2].nGood) + DINT_TO_REAL(stStatisticsHMI[2].nBad))) * 100.0,iPrecision := 2, bRound := TRUE);
	stStatisticsHMI[2].nEfficency		:= CONCAT(STR1 := '%', STR2 := (rEfficency));

ELSE stStatisticsHMI[2].nEfficency		:= CONCAT(STR1 := '%', STR2 := (DINT_TO_STRING(0)));
	
END_IF
END_ACTION

ACTION d_ACT_Set_Events_Station_2:
//IMMEDIATE FAULTS

stStationEvents[2].aEvents[0].bImmediateFault				:= TRUE;
stStationEvents[2].aEvents[0].bEventFlag					:= bEventsFlag[0];
stStationEvents[2].aEvents[0].bEventText					:= 'ST1 EVENT 0';
stStationEvents[2].aEvents[0].sSolution						:= 'Solution 3';


//CYCLE STOP FAULT

stStationEvents[2].aEvents[1].bCycleStopFault				:= TRUE;
stStationEvents[2].aEvents[1].bEventFlag					:= bEventsFlag[1];
stStationEvents[2].aEvents[1].bEventText					:= 'ST1 EVENT 1';
stStationEvents[2].aEvents[1].sSolution						:= 'Solution 4';


//CYCLE STOP REQUEST

stStationEvents[2].aEvents[2].bCycleStopRequest			:= TRUE;
stStationEvents[2].aEvents[2].bEventFlag					:= bEventsFlag[2];
stStationEvents[2].aEvents[2].bEventText					:= 'ST1 EVENT 2';
END_ACTION

END_PROGRAM

// ---- POUs/Utilities/FB_WriteDataToCSV.TcPOU
FUNCTION_BLOCK FB_WriteDataToCSV
VAR_INPUT
	
	bWriteCSV		: BOOL;(* Rising edge starts program execution *)
	bWriteData		: BOOL;
	sFileNamePath	: STRING(255);
	aDataHistory	: ARRAY[0..200] OF ST_EventsHistory;
	aDataHistoryArrayLength : DINT;
	sDate			: STRING(255);
	
	nMAX_CSV_ROWS	: UDINT;
	nMAX_CSV_COLUMNS: UDINT;
	

END_VAR
VAR_OUTPUT
	
	bBusy			: BOOL;
	bError			: BOOL;
	nErrId			: UDINT;
	
END_VAR
VAR
	
	
	sCSVField		: T_MaxString := '';(* Single CSV field value (column, record field) *)
	nRow	 		: UDINT 	:= 0;(* Row number (record) *)
	nColumn			: UDINT 	:= 0;(* Column number (record field) *)
	hFile			: UINT		:= 0;(* File handle of the source file *)
	step			: DWORD 	:= 0;
	fbFileOpen		: FB_FileOpen;(* Opens file *)
	fbFileClose		: FB_FileClose;(* Closes file *)
	fbFilePuts		: FB_FilePuts;(* Writes one record (line) *)
	fbWriter		: FB_CSVMemBufferWriter;(* Helper function block used to create CSV data bytes (single record line) *)
	sCSVLine		: T_MaxString := '';(* Single CSV text line (row, record), we are using string as record buffer (your are able to see created fields) *)
	database		: ARRAY[0..10000(*MAX ROWS*), 0..(*MAX COLUMS*)6] OF STRING(255(*MAX STRING LENGTH*));
	nRowIndex		: DINT;
	i				: DINT;
	sCSVDate		: STRING(255);
	bFirstScan		: BOOL;
	rWriteCSV		: R_TRIG;
	rWriteData		: R_TRIG;
	
	sFileName		: T_MaxString ;(* CSV destination file path and name *)
	
	
END_VAR
VAR_IN_OUT

END_VAR

//TO USE THIS FUNCTION DEFINE "MAX ROWS", "MAX COLUMS" AND "MAX STRING LENGTH". THEY SHOULD BE EQUAL TO INPUTS

ACT_Write();
ACT_CSVSettings();


rWriteData( CLK := bWriteData);

IF NOT bFirstScan THEN
	
	sCSVDate								:= sDate;
	bFirstScan								:= TRUE;

END_IF

ACTION ACT_CSVSettings:

IF sCSVDate <> sDate THEN
	
	sCSVDate							:= sDate;

END_IF

sFileName 								:= CONCAT(sFileNamePath,CONCAT( STR1 := '_', STR2 := CONCAT( STR1:= sCSVDate, STR2 := '.csv')));


IF rWriteData.Q THEN
	
	FOR i := 0 TO aDataHistoryArrayLength DO
		
		IF aDataHistory[i].sEventTex <> '' THEN
			
					database[nRowIndex,0]				:= 	aDataHistory[i].sEventTex;
					database[nRowIndex,1]				:= 	aDataHistory[i].sType;
					database[nRowIndex,2]				:= 	aDataHistory[i].sDate;
					database[nRowIndex,3]				:= 	aDataHistory[i].sTime;
					nRowIndex							:= nRowIndex + 1;
		END_IF
					

				
	END_FOR
	
	i													:= 0;

	

END_IF
END_ACTION

ACTION ACT_Write:
rWriteCSV( CLK := bWriteCSV);
CASE step OF
	0:	(* Wait for rising edge at bWrite variable *)
		IF rWriteCSV.Q THEN
				
			bBusy 	:= TRUE;
			bError	:= FALSE;
			nErrId	:= 0;
			hFile	:= 0;
			nRow	:= 0;
			nColumn	:= 0;
			step 	:= 1;

		END_IF

	1:	(* Open source file *)
		fbFileOpen(  bExecute := FALSE  );
		fbFileOpen( sNetId := NetAmsId , sPathName := sFileName, nMode := FOPEN_MODEWRITE OR FOPEN_MODETEXT,(* Open file in TEXT mode! *)
					ePath := PATH_GENERIC, bExecute := TRUE );
		step := 2;

	2:(* Wait until open not busy *)
		fbFileOpen( bExecute := FALSE, bError => bError, nErrID => nErrID, hFile => hFile );
		IF NOT fbFileOpen.bBusy THEN
			IF NOT fbFileOpen.bError THEN
				step := 3;
			ELSE(* Error: file not found? *)
				step := 100;
			END_IF
		END_IF

	3:(* Convert one PLC record to CSV format *)
		sCSVLine := '';
		fbWriter.eCmd := eEnumCmd_First;(* Write first field value *)
		IF nRow <= nMAX_CSV_ROWS THEN

			FOR nColumn := 0 TO nMAX_CSV_COLUMNS BY 1 DO

				sCSVField := STRING_TO_CSVFIELD( database[ nRow, nColumn ], FALSE );(* TODO: Get field value from your application *)

				(* Add new field to the record buffer *)
				fbWriter( 	pBuffer := ADR( sCSVLine ), cbBuffer := SIZEOF( sCSVLine ) - 1, putValue := sCSVField, pValue := 0, cbValue := 0(*,
							bCRLF := ( nColumn = nMAX_CSV_COLUMNS )*) );(* bCRLF == TRUE => Write CRLF after the last field value *)
				IF fbWriter.bOk THEN
					fbWriter.eCmd := eEnumCmd_Next;(* Write next field value *)
				ELSE(* Error *)
					step := 100;
					RETURN;
				END_IF
				
			END_FOR(* FOR nColumn := 0... *)

			(* FB_FilePuts adds allready CR (carriage return) to the written line.
			We have to replace the $R$L characters with $L character to avoid double CR. *)
			IF RIGHT( sCSVLine, 2 ) = '$R$L' THEN
				sCSVLine := REPLACE( sCSVLine, '$L', 2, LEN( sCSVLine ) - 1 );
			END_IF

			nRow := nRow + 1;(* Increment number of created records (rows) *)
			step := 4;(* Write record to the file *)

		ELSE(* All rows written => Close file *)
			step := 10;
		END_IF

	4:	(* Write single text line *)
		fbFilePuts( bExecute := FALSE );
		fbFilePuts( sNetId := NetAmsId , hFile := hFile, sLine := sCSVLine, bExecute := TRUE );
		step := 5;

	5:(* Wait until write not busy *)
		fbFilePuts( bExecute := FALSE, bError => bError, nErrID => nErrID );
		IF NOT fbFilePuts.bBusy THEN
			IF NOT fbFilePuts.bError THEN
				step := 3;(* Write next record *)
			ELSE(* Error *)
				step := 100;
			END_IF
		END_IF

	10:	(* Close source file *)
		fbFileClose( bExecute := FALSE );
		fbFileClose( sNetId := NetAmsId , hFile := hFile, bExecute := TRUE );
		step := 11;

	11:(* Wait until close not busy *)
		fbFileClose( bExecute := FALSE, bError => bError, nErrID => nErrID );
		IF ( NOT fbFileClose.bBusy ) THEN
			hFile := 0;
			step := 100;
		END_IF

	100: (* Error or ready step => cleanup *)
		IF ( hFile <> 0 ) THEN
			step := 10; (* Close the source file *)
		ELSE
			bBusy := FALSE;
			step := 0;	(* Ready *)
		END_IF

END_CASE
END_ACTION

END_FUNCTION_BLOCK
